# EPICS IOC start-up script: examples/test/PSI/EP6224/EP6334_MurrEmparro67.iocsh
#- #############################################################################
#- mXsXXX naming
require ecmccfg v7_RC1, "ECMC_VER=dev,NAMING=mXsXXX,MASTER_ID=0"

#- #############################################################################
#- add slaves
${SCRIPTEXEC} ${ECMC_CONFIG_ROOT}addSlave.cmd, "HW_DESC=EP6224, SLAVE_ID=${SLAVE=0}"
${SCRIPTEXEC} ${ECMC_CONFIG_ROOT}applySlaveConfig.cmd, "CONFIG=-Sensor-Murr-emparro67, ECMC_EC_CH_ID=4"
${SCRIPTEXEC} ${ECMC_CONFIG_ROOT}applySubstitutions.cmd, "SUBST_FILE=./Emparro67.subs"

#- #############################################################################
#- apply hardware configuration
${SCRIPTEXEC} ${ecmccfg_DIR}applyConfig.cmd

#- #############################################################################
#- configure diagnostics
ecmcConfigOrDie "Cfg.EcSetDiagnostics(1)"
ecmcConfigOrDie "Cfg.EcEnablePrintouts(0)"
ecmcConfigOrDie "Cfg.EcSetDomainFailedCyclesLimit(100)"

# go active
${SCRIPTEXEC} ${ecmccfg_DIR}setAppMode.cmd
#- #############################################################################
